// TIA Portal V19 export
DATA_BLOCK "Gestion des sorties MANU_DB"   // DB11
// stored: InstanceOfName Gestion des sorties, InstanceOfType FB
"Gestion des sorties"
BEGIN
END_DATA_BLOCK
